ABB RobotStudio station: NewNewStation.rspag

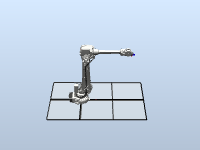
--- station ---
Station Station (saved by RobotStudio format 3)
Controller NewNewSystem
  mechanical unit ROB_1: IRB4600_40_255_C_01, 6 joints, base frame (0, 0, 0) mm
Layout (positions relative to the parent item):
  - IRB4600_40_255_C_01 [mechanism, from Robots\IRB4600_40_255_C_G_01.rslib] at (0, 0, 0) mm; joint values [0, 0, 0, 0, 0.5236, 0] (rad or m)

--- Backups/NewNewSystem/RAPID/TASK1/PROGMOD/RRI_newmodule.mod ---
MODULE RRI_newmodule
    RECORD robotdata
        num type;
        string status;
    ENDRECORD

    RECORD replydata
        num type;
        string status;
!        string Mode;
        num Time;
    ENDRECORD

    PERS sensor TestDevice := [-1,2602,-1];
    PERS robotdata RobotMessage := [0,""];
    PERS replydata ReplyMessage := [34,"",23];


    PROC Main()
    SiConnect TestDevice;
    SiSetCyclic TestDevice, RobotMessage, 800;
    SiGetCyclic TestDevice, ReplyMessage, 800;

!    TPWrite "ReplyMessage " \Num:=ReplyMessage;
    ENDPROC

ENDMODULE

--- Backups/NewNewSystem/SYSPAR/EIO.cfg ---
EIO:CFG_1.0:5:60::
#
EIO_BUS:

      -Name "Virtual1" -ConnectorID "SIM1"
#
EIO_UNIT_TYPE:

      -Name "Virtual" -VendorName "ABB" -ProductName "Virtual unit"
#
EIO_ACCESS:

      -Name "All" -Rapid  -LocalManual  -LocalAuto  -RemoteManual  -RemoteAuto
